Universal Robots URScript: 00B_02_JuXian.script

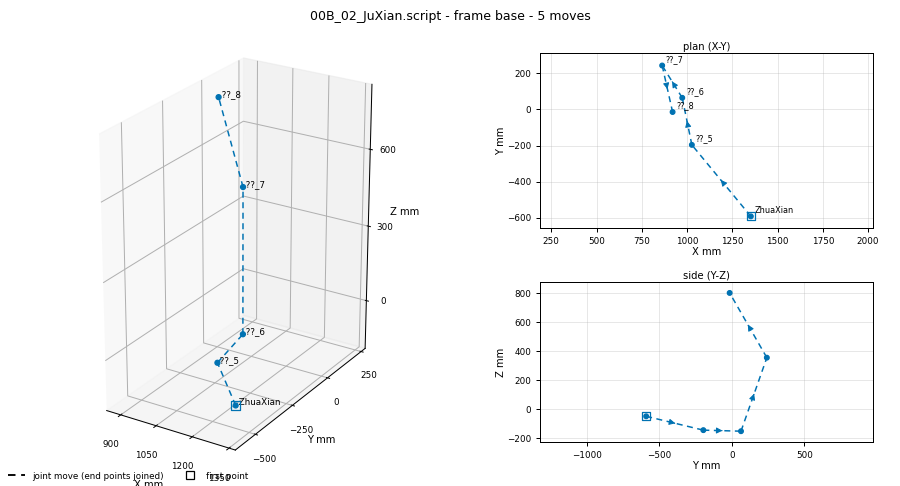
[picture p0: tool path of 00B_02_JuXian.script in frame base, 5 of 5 moves have a stored position in this frame; points joined in program order, loops and branches not executed]
def P00B_02_JuXian():
  set_gravity([0.0, 0.0, 9.82])
  set_safety_mode_transition_hardness(1)
  set_standard_analog_input_domain(0, 1)
  set_standard_analog_input_domain(1, 1)
  set_tool_analog_input_domain(0, 1)
  set_tool_analog_input_domain(1, 1)
  set_analog_outputdomain(0, 0)
  set_analog_outputdomain(1, 0)
  set_tool_voltage(24)
  set_input_actions_to_default()
  set_tcp(p[0.0,0.0,0.32,0.0,0.0,-0.5236])
  set_payload(8.0)
  global Zhua_1=[0.08063, -2.42649, -1.72682, -0.47876, 0.40808, -1.10831]
  global prepose=p[0.98979, -0.16931, -0.39963, 1.98720, 0.07234, 0.05469]
  global i_var_2=0
  global i_var_1=True
  global pose=p[0.98979, -0.31931, -0.39963, 1.98720, 0.07234, 0.05469]
  $ 1 "机器人程序"
  $ 2 "MoveJ"
  $ 3 "ZhuaXian"
  set_tcp(p[0.0,0.0,0.32,0.0,0.0,-0.5236])
  movej(get_inverse_kin(p[1.352436109272, -.591216839006, -.049372824621, .134324829362, 1.558483226668, -.012546260116], qnear=[-0.4123619238482874, -2.654867474232809, -1.1444781462298792, -2.4834540526019495, -1.8943169752704065, -0.9837244192706507]), a=0.6981317007977318, v=0.5235987755982988)
  $ 4 "路点_5"
  set_tcp(p[0.0,0.0,0.32,0.0,0.0,-0.5236])
  movej(get_inverse_kin(p[1.026681930282, -.196415542214, -.145098439602, .158376044317, 1.750934500312, -.000171896431], qnear=[0.013871366158127785, -2.237016503010885, -2.1720269362079065, -2.0628965536700647, -1.4715130964862269, -0.9471319357501429]), a=0.6981317007977318, v=0.5235987755982988)
  $ 5 "路点_6"
  set_tcp(p[0.0,0.0,0.32,0.0,0.0,-0.5236])
  movej(get_inverse_kin(p[.973614045542, .063507284781, -.152369900391, -.043710575992, 1.815017474621, .606270674040], qnear=[0.013883350417017937, -2.23702842393984, -2.171882931386129, -2.104039494191305, -1.9967358748065394, -0.7533100287066858]), a=0.6981317007977318, v=0.5235987755982988)
  $ 6 "路点_7"
  set_tcp(p[0.0,0.0,0.32,0.0,0.0,-0.5236])
  movej(get_inverse_kin(p[.862738274729, .241895799601, .355282502729, .664557731137, 1.544631161189, 1.007345205343], qnear=[0.7286427617073059, -1.299699608479635, -2.2724931875811976, -2.725281063710348, -1.087172810231344, 0.011706715449690819]), a=0.6981317007977318, v=0.5235987755982988)
  $ 7 "路点_8"
  set_tcp(p[0.0,0.0,0.32,0.0,0.0,-0.5236])
  movej(get_inverse_kin(p[.920290202912, -.014783162077, .802161983438, 1.103598835514, 1.210552194825, 1.370150264948], qnear=[0.19962535798549652, -1.2916463057147425, -1.5798857847796839, -3.315007988606588, -1.4863570372210901, 0.5352832674980164]), a=0.6981317007977318, v=0.5235987755982988)
end
